// Mitsubishi GX Works2 project: 컨베이어벨트 LED 0906   PLC: Q03UDV

PROGRAM MAIN
VAR
  TOK30 : BOOL;
END_VAR
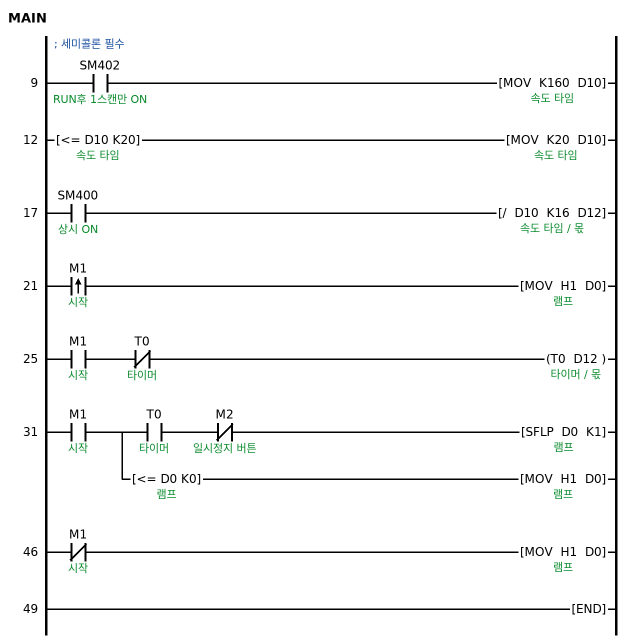
; 세미콜론 필수
9     LD      SM402  ; RUN후 1스캔만 ON
      MOV     K160 D10  ; 속도 타임
12    LD<=    D10 K20  ; 속도 타임
      MOV     K20 D10
17    LD      SM400  ; 상시 ON
      /       D10 K16 D12  ; 몫
21    LDP     M1  ; 시작
      MOV     H1 D0  ; 램프
25    LD      M1  ; 시작
      ANI     T0  ; 타이머
      OUT     T0 D12  ; 타이머 / 몫
31    LD      M1  ; 시작
      MPS
      AND     T0  ; 타이머
      ANI     M2  ; 일시정지 버튼
      SFLP    D0 K1
      MPP
      AND<=   D0 K0  ; 램프
      MOV     H1 D0
46    LDI     M1  ; 시작
      MOV     H1 D0
49    END
END_PROGRAM

// device comments not shown above
M0  ; 초기화
M10  ; 패킹 ON
Y10  ; RL램프
Y11  ; 램프2
Y40  ; 램프
D1  ; 패킹 단위
D2  ; 패킹 수량
